{attribute addProperty BoxType "EL5151-0021-0018"}
{attribute addProperty Id "Latch_C_validBIT10.1251Latch_extern_validBIT10.1252Set_counter_doneBIT10.1253Measurement_doneBIT10.1252Status_of_input_ABIT10.1259Status_of_input_BBIT10.12510Status_of_input_CBIT10.12511Status_of_outputBIT10.1251Status_of_extern_latchBIT10.12513Compatible_input_cycle_counter_highBIT10.12514TxPDO_ToggleBIT10.12516"}
{attribute addProperty CRC "1426574155"}
{attribute addProperty SizeInBites "16"}
{attribute addProperty SizeInBytes "2"}
TYPE Status_5507CB4B :
STRUCT
	{attribute addProperty Name "Latch_C_valid"}
	Latch_C_valid : BIT;
	{attribute addProperty Name "Latch_extern_valid"}
	Latch_extern_valid : BIT;
	{attribute addProperty Name "Set_counter_done"}
	Set_counter_done : BIT;
	{attribute 'hide'}
	reserve_1_BIT_0 : BIT;
	{attribute 'hide'}
	reserve_1_BIT_1 : BIT;
	{attribute addProperty Name "Measurement_done"}
	Measurement_done : BIT;
	{attribute 'hide'}
	reserve_2_BIT_0 : BIT;
	{attribute 'hide'}
	reserve_2_BIT_1 : BIT;
	{attribute addProperty Name "Status_of_input_A"}
	Status_of_input_A : BIT;
	{attribute addProperty Name "Status_of_input_B"}
	Status_of_input_B : BIT;
	{attribute addProperty Name "Status_of_input_C"}
	Status_of_input_C : BIT;
	{attribute addProperty Name "Status_of_output"}
	Status_of_output : BIT;
	{attribute addProperty Name "Status_of_extern_latch"}
	Status_of_extern_latch : BIT;
	{attribute addProperty Name "Compatible_input_cycle_counter_high"}
	Compatible_input_cycle_counter_high : BIT;
	{attribute 'hide'}
	reserve_3 : BIT;
	{attribute addProperty Name "TxPDO_Toggle"}
	TxPDO_Toggle : BIT;
END_STRUCT
END_TYPE

(* stored: Version 1.2.0.0, ProductVersion 3.1.4024.9
   DUT Status_5507CB4B: Id {489251f1-ad60-415a-92ff-deaec8f37d5f} *)
